// TIA Portal V20 export
FUNCTION_BLOCK "FB_Part_Data"   // FB93, SCL
{ S7_Optimized_Access := 'TRUE' }
// stored: MemoryReserve 100, SetENOAutomatically false
   VAR
      Part_Data_Ident : "FB_ReadWrite_GUDs";
      sWriteDataEnable { S7_SetPoint := 'True'} : Bool;
      sNewPartDataIdent : Bool;
      RT_NewPartDataIdent : R_TRIG;
      sCurrentPartDataIdent { S7_SetPoint := 'True'} : String;
   END_VAR
   VAR_TEMP
      tIndex : Int;
   END_VAR
BEGIN
   REGION Description header 
       //==================================================================================
       // POSALUX Swiss SA / (C) Copyright 2026
       //----------------------------------------------------------------------------------
       // Title: FB_Part_Data
       // Comment/Function: 
       //
       // Author: Fabien WALDT
       // Engineering: TIA Portal v20
       //----------------------------------------------------------------------------------
       // Change log table:
       // Version  | Date     | Expert in charge | Changes applied
       // ---------|----------|------------------|------------------------------------
       // 00.00.01 | 20260518 | WFA              | First released version
       // ==================================================================================
   END_REGION

   REGION Data Init
       #Part_Data_Ident.sName := 'PART_DATA_IDENT';
       #Part_Data_Ident.sType := 4;
       #Part_Data_Ident.sNCK_channel := 1;
    //   #Part_Data_Ident.sWriteVal_String[0] := 'Test_ID_From_PLC';
   END_REGION

   REGION Call Read/Wrtite GUD
       #Part_Data_Ident();
   END_REGION

   REGION Convert DMC into String

   END_REGION

   REGION New Value
   // Convert DMC Array into String    
   Chars_TO_Strg(Chars:= "DB_DataPositions".Position[4].DMC,
                 pChars:= 0,
                 Cnt:= 19,
                 Strg=> #sCurrentPartDataIdent);

   // Check if new Part on Fixture
   IF #Part_Data_Ident.sWriteVal_String[0] <> #sCurrentPartDataIdent THEN
       #Part_Data_Ident.sWriteVal_String[0] := #sCurrentPartDataIdent;
       #sNewPartDataIdent := TRUE;
       END_IF;
   END_REGION

   // Il faut tout d'abord effectuer une lecture :
   // #Part_Data_Ident.sStart_rd
   // Pour obtenir #Part_Data_Ident.sRead_done
   // On peut alors effctuer une ecriture avec #Part_Data_Ident.sStart_wr
   // Pour obtenir #Part_Data_Ident.sWrite_done

   REGION Write Datas Request
       IF NOT #sWriteDataEnable THEN
           #Part_Data_Ident.sStart_rd := TRUE;
       END_IF;

   IF #Part_Data_Ident.sRead_done THEN
       #Part_Data_Ident.sStart_rd := FALSE;
       #sWriteDataEnable := TRUE;
   END_IF;

   #RT_NewPartDataIdent(CLK := #sNewPartDataIdent);
   IF #RT_NewPartDataIdent.Q AND #sWriteDataEnable THEN
       #Part_Data_Ident.sStart_wr := TRUE;
       #sNewPartDataIdent := FALSE;
   ELSIF #Part_Data_Ident.sWrite_done THEN
       #Part_Data_Ident.sStart_wr := FALSE;
   END_IF;
   END_REGION
END_FUNCTION_BLOCK
